// TIA Portal V17 export
BLOCK "FC_Compare"   // ObjectSW15, LAD
BEGIN

REGION Network 1: compare chain
END_REGION
END_BLOCK
